{attribute 'linkalways'} 
{attribute 'no_explicit_call' := 'This FB is a CLASS and must be accessed using methods or properties'}
{attribute 'enable_dynamic_creation'}
FUNCTION_BLOCK _TcVnParamsKAZE EXTENDS StructuredDatatypeBase
VAR
	localData : TcVnParamsKAZE;
	activeData : REFERENCE TO TcVnParamsKAZE REF= localData;
    _bExtended     : _BOOL(localdata.bExtended);
    _bUpright      : _BOOL(localdata.bUpright);
    _fThreshold    : _REAL(localdata.fThreshold);
    _nOctaves      : _UDINT(localdata.nOctaves);
    _nOctaveLayers : _UDINT(localdata.nOctaveLayers);
    _eDiffusivity  : _ETcVnDiffusivityTypeKAZE(localdata.eDiffusivity);
END_VAR

PROPERTY PUBLIC Address : PVOID
GET
Address := ADR(activeData);
END_GET
END_PROPERTY

PROPERTY PUBLIC bExtended : REFERENCE TO _BOOL
GET
bExtended REF= _bExtended;
END_GET
END_PROPERTY

PROPERTY PUBLIC bUpright : REFERENCE TO _BOOL
GET
bUpright REF= _bUpright;
END_GET
END_PROPERTY

METHOD PUBLIC ClearReference
VAR_INPUT
END_VAR
activeData REF= localData;
SetMemberReference();
END_METHOD

METHOD PUBLIC Clone : I_Datatype
VAR
    pClone : POINTER TO _TcVnParamsKAZE;
END_VAR
pClone := __NEW(_TcVnParamsKAZE());
pClone^.Value := Value;
Clone := pClone^;
END_METHOD

PROPERTY PUBLIC eDiffusivity : REFERENCE TO _ETcVnDiffusivityTypeKAZE
GET
eDiffusivity REF= _eDiffusivity;
END_GET
END_PROPERTY

METHOD FB_init : BOOL
VAR_INPUT
	bInitRetains : BOOL; // if TRUE, the retain variables are initialized (warm start / cold start)
	bInCopyCode : BOOL;  // if TRUE, the instance afterwards gets moved into the copy code (online change)
END_VAR
SetMemberReference();
AddMember('bExtended', _bExtended);
AddMember('bUpright', _bUpright);
AddMember('fThreshold', _fThreshold);
AddMember('nOctaves', _nOctaves);
AddMember('nOctaveLayers', _nOctaveLayers);
AddMember('eDiffusivity', _eDiffusivity);
END_METHOD

PROPERTY PUBLIC fThreshold : REFERENCE TO _REAL
GET
fThreshold REF= _fThreshold;
END_GET
END_PROPERTY

PROPERTY PUBLIC Identifier : T_MAXSTRING
GET
Identifier := 'TcVnParamsKAZE';
END_GET
END_PROPERTY

METHOD PUBLIC MakeReferenceTo
VAR_INPUT
	ReferenceTarget : REFERENCE TO TcVnParamsKAZE;
END_VAR
activeData REF= ReferenceTarget;
SetMemberReference();
END_METHOD

PROPERTY PUBLIC nOctaveLayers : REFERENCE TO _UDINT
GET
nOctaveLayers REF= _nOctaveLayers;
END_GET
END_PROPERTY

PROPERTY PUBLIC nOctaves : REFERENCE TO _UDINT
GET
nOctaves REF= _nOctaves;
END_GET
END_PROPERTY

METHOD PROTECTED SetMemberReference
VAR_INPUT
END_VAR
_bExtended.MakeReferenceTo(activeData.bExtended);
_bUpright.MakeReferenceTo(activeData.bUpright);
_fThreshold.MakeReferenceTo(activeData.fThreshold);
_nOctaves.MakeReferenceTo(activeData.nOctaves);
_nOctaveLayers.MakeReferenceTo(activeData.nOctaveLayers);
_eDiffusivity.MakeReferenceTo(activeData.eDiffusivity);
END_METHOD

PROPERTY PUBLIC Size : UDINT
GET
Size := SIZEOF(activeData);
END_GET
END_PROPERTY

METHOD TryMakeReferenceTo : BOOL
VAR_INPUT
	Target : I_Datatype;
END_VAR
VAR
	pTargetData : POINTER TO TcVnParamsKAZE;
END_VAR
IF NOT IsEquivalentTo(Target) THEN
	RETURN;
END_IF

pTargetData := Target.Address;
activeData REF= pTargetData^;
SetMemberReference();
TryMakeReferenceTo := TRUE;
END_METHOD

PROPERTY PUBLIC Value : REFERENCE TO TcVnParamsKAZE
GET
Value REF= activeData;
END_GET
END_PROPERTY

END_FUNCTION_BLOCK

(* stored: Version 1.1.0.1, ProductVersion 3.1.4024.13
   POU _TcVnParamsKAZE: Id {1089b0e5-6e90-0d57-05f9-827cd041328a}, SpecialFunc None
   Folder Core: Id {dbc8acb4-4db7-008f-060e-74332a172dd1}
   Folder Customize: Id {270c0b63-d7f4-0479-29af-baec9ead84fe}
   Folder Constructor: Id {6b3d1f82-27df-0405-167a-135e57fa40e0}
   Folder Protected: Id {5723b9bf-e367-0aeb-3f54-4135c2e8f14b}
   Property Address: Id {a5418e27-5a6f-0740-02a2-3989c436e92d}
   Get Get: Id {f83852e7-12dc-04e5-36ec-bb3e995e6580}
   Property bExtended: Id {cf28a7e7-158b-0503-2c25-d58ff2c1f3bf}
   Get Get: Id {5cfca72c-2b12-0449-33c1-fa5674218b49}
   Property bUpright: Id {69bde511-4763-05a2-0560-086b5366625c}
   Get Get: Id {f4ae5ab3-ee73-0550-0cfc-f57d716aa0d2}
   Method ClearReference: Id {0abc11f2-00ac-0200-2a67-71105a654838}
   Method Clone: Id {bbd263c6-2d33-03e5-1ad2-ae1cfa04747f}
   Property eDiffusivity: Id {e69d658b-387b-0347-15ee-8ca8219368ef}
   Get Get: Id {3c9d96ea-08f6-0407-242f-bde505323e0c}
   Method FB_init: Id {075fa414-2fe7-0e1f-29d9-67cf1c03c796}
   Property fThreshold: Id {338733ac-0fba-059f-2bc0-8093fa929b37}
   Get Get: Id {10dd2f1f-ec6b-0f9d-1612-a79de9118aa1}
   Property Identifier: Id {5a9ad19e-d913-074f-0a19-ee307e846a87}
   Get Get: Id {bf7febe8-9bae-0295-2bb2-5705410208e7}
   Method MakeReferenceTo: Id {8a7b3470-84e6-05c9-370d-71a165780947}
   Property nOctaveLayers: Id {5f182217-930d-0f83-3b91-bf75e380dd64}
   Get Get: Id {26fc345b-9758-0f4f-1448-5d7d9bf418af}
   Property nOctaves: Id {7e8396e2-9414-0ed8-0547-e38cdfc1814c}
   Get Get: Id {cc0350ac-58ad-0698-1cab-89151c04d4bc}
   Method SetMemberReference: Id {5c019f7c-0134-0dda-204c-0ec2902443d2}
   Property Size: Id {22a77cfb-03e4-0857-226f-54c303c6db2c}
   Get Get: Id {a6245898-6dbc-0c7d-13fa-73008173f033}
   Method TryMakeReferenceTo: Id {27f681ad-d569-08e7-12e7-c910c5dfc63e}
   Property Value: Id {ee6367fe-2e44-0ed0-020c-d9afcba7eb36}
   Get Get: Id {47f8f709-8410-0dfd-37c6-e07e7de5c75a} *)
